// TIA Portal V20 export
// export: Created 2026-04-10T22:01:57.8449221Z, ExportSetting WithDefaults, DisplayName Totally Integrated Automation Portal, DisplayVersion V20, DisplayName TIA Portal Openness, DisplayVersion V20, DisplayName TIA Portal Version Control Interface, DisplayVersion V20, DisplayName STEP 7 Professional, DisplayVersion V20, DisplayName STEP 7 Safety, DisplayVersion V20, DisplayName WinCC Basic/Comfort/Advanced, DisplayVersion V20
VAR_GLOBAL   // PLC tag table "MES_"
END_VAR
VAR_GLOBAL CONSTANT   // user constants
   MES_CommunicationError : Int := 1;   // Kommentar MES_CommError
   MES_BLOCKED : Int := 2;   // Kommentar MES_BLOCKED
   MES_TRANSFER_FAILED : Int := 3;   // Kommentar MES_TRANSFER_FAILED
END_VAR
